FUNCTION_BLOCK FB_AUT_140 EXTENDS FB_AUT_ABSTRACT
(****************************************************************************)
(*	POU_AUT_zxx			Bausteinaufrufe Station	zxx							*)
(*	Status				ungetestet											*)
(*  Version:			1.0													*)
(*	Beschrieb:																*)
(*																			*)
(*	Abläufe:			FB_ABLzxxA		Hauptablauf							*)
(*																			*)
(*																			*)
(* 	25.09.2019/Dj															*)
(****************************************************************************)
(*	dd.mm.yyyy   KZ    x.y			Beschrieb								*)
(****************************************************************************)
VAR_INPUT
    (* spezifische Eingänge *)

END_VAR
VAR_OUTPUT
    (* spezifische Ausgänge *)

END_VAR
VAR
    (* Bausteine *)
    fb_Measure : FB_ABL_140_Measure;

END_VAR

(*******************************************************************)
(* Timer *)
(*******************************************************************)

(*******************************************************************)
(* Flanken / Merker *)
(*******************************************************************)
//MANU CYCLE
IF (enIN_State = StateMANU) AND xIN_ManuCycle THEN
    xManuCycle := TRUE;
END_IF;

IF (enIN_State <> StateMANU) OR xOUT_Done THEN
    xManuCycle := FALSE;
END_IF

//NEXT STEP
xNextStep := (enIN_State > StateSTEP) OR
             ((enIN_State = StateSTEP) AND xIN_Step) OR
             ((enIN_State = StateMANU) AND xManuCycle);

//RESET
xReset := (enIN_State < StateREADY) AND (enIN_State <> StateINIT) AND NOT xManuCycle;

(*******************************************************************)
(* Bausteinaufrufe Abläufe *)
(*******************************************************************)

fb_Measure(xIN_Reset          := xReset,
       xIN_Init           := xIN_Init,
       xIN_Quit           := xIN_Quit,
       xIN_Start          := enIN_State = enState.StateAUTO, //AND _FB_ABL_100A.xOUT_Done AND _FB_ABL_100A.xOUT_Ready,
       xIN_Sperre         := NOT xIN_On,
       xIN_NextStep       := xNextStep,
       xIN_AlarmAktiv     := xIN_AlarmAktiv,
       xIN_DryCycle       := xIN_DryCycle,
       xIN_RestartCYCL    := enIN_State = enState.StateAUTO, // only restart when the mover has move out
       enIN_State         := enIN_State,
       tIN_Timeout        := tIN_Timeout,
       pxFG_Freigabe      := ADR(xDummy),
       Mover              := THIS^.Mover);

(*******************************************************************)
(* Mover reset flags *)
(*******************************************************************)

(*******************************************************************)
(* OUTPUT *)
(*******************************************************************)
xOUT_InitDone := fb_Measure.xOUT_InitDone;
xOUT_Ready    := fb_Measure.xOUT_Ready;
xOUT_Done     := fb_Measure.xOUT_Done;
xOUT_ErrFlag  := fb_Measure.xOUT_ErrFlag;
xOUT_Wait     := fb_Measure.xOUT_Wait;
xOUT_AlarmST  := xOUT_ErrFlag;

(*******************************************************************)
(* Bausteinaufruf Error Station *)
(*******************************************************************)
// POU_ERR_VORLAGE(xIN_QUIT:=xIN_Quit , pstrArIN_ALARM:=ADR(HMI.strArALARM[1]));

(* % of completion of the process *)
PROPERTY iCompletionPC : INT
GET
iCompletionPC := THIS^.fb_Measure.iOUT_ProcessCompletion;
END_GET
END_PROPERTY

PROPERTY ProcessExecution : ProcessExecution_e
GET
ProcessExecution := THIS^._ProcessExecution;
END_GET
SET
THIS^._ProcessExecution := ProcessExecution;
END_SET
END_PROPERTY

PROPERTY xBusy : BOOL
GET
xBusy := THIS^.fb_Measure.xOUT_Busy;
END_GET
SET
END_SET
END_PROPERTY

PROPERTY xDone : BOOL
GET
xDone := THIS^.fb_Measure.xOUT_Ready OR THIS^.fb_Measure.xOUT_Done;
END_GET
END_PROPERTY

PROPERTY xMoverPathFree : BOOL
GET
xMoverPathFree := THIS^.fb_Measure.xOUT_MoverFree OR THIS^.fb_Measure.xOUT_Ready OR THIS^.fb_Measure.xOUT_Done;
END_GET
END_PROPERTY

PROPERTY xMoverShouldLeave : BOOL
GET
xMoverShouldLeave := THIS^.fb_Measure.iOUT_Step = ST140_Measure_e.SYNC_MOVER_LEAVE;
END_GET
END_PROPERTY

END_FUNCTION_BLOCK

(* stored: Version 1.1.0.1, ProductVersion 3.1.4024.6
   POU FB_AUT_140: Id {b97e51aa-fc97-4727-93f4-9bc927d088d5}, SpecialFunc None
   Property iCompletionPC: Id {dd467b5e-e5e2-4ebd-9c80-0c080b3207f7}
   Get Get: Id {8db43e4b-91d2-4382-bbac-6d5eca4ebb18}
   Property ProcessExecution: Id {a2dd3edb-082b-4dd4-b929-042ab0faae70}
   Get Get: Id {926ff66c-80b2-4019-8e38-c790b73bb361}
   Set Set: Id {d91c7029-cdd2-4c63-a646-80d337b30696}
   Property xBusy: Id {fa7b9acf-77d7-4703-9b62-9928c4d9294f}
   Get Get: Id {5ef03455-4074-4163-9f8f-725e120501e2}
   Set Set: Id {5d75f20d-8d4a-4112-ae6e-9d22bd0e9b18}
   Property xDone: Id {44bd8c8c-24dc-4756-9384-c98760dd892b}
   Get Get: Id {4f1c4da4-c4bd-40ae-b1c3-24d01a7d244d}
   Property xMoverPathFree: Id {e5473a74-874a-4720-ab76-e3020920437a}
   Get Get: Id {118019a3-0683-41e8-86c3-6b65fc9bfbb3}
   Property xMoverShouldLeave: Id {00fc1311-c71b-470a-b30b-be3d4a56a97f}
   Get Get: Id {fa4f73e1-0dd7-4eb7-9b9b-e3e6cfa9d84d} *)
